{attribute 'GeneratedUsingTerminal: EL5001--0000'}
{attribute addProperty BoxType "EL5001--0000"}
{attribute addProperty Description "EL5001 1Ch. SSI Encoder"}
{attribute addProperty Physics "KK"}
{attribute addProperty Id "Channel_1AT %I*Channel_4E63E14D5WcStateAT %I*WcState_9091E0EB2InfoDataAT %I*InfoData_32EB74EA10"}
{attribute addProperty CRC "1375238614"}
{attribute addProperty Size "17"}
TYPE EL5001_51F879D6 EXTENDS EtcSlaveTerminalBase_947E5A46 :
STRUCT
	{attribute addProperty Name "Channel_1"}
	Channel_1 : Channel_4E63E14D;
	{attribute addProperty Name "WcState"}
	WcState : WcState_9091E0EB;
	{attribute addProperty Name "InfoData"}
	InfoData : InfoData_32EB74EA;
END_STRUCT
END_TYPE

(* stored: Version 1.2.0.0, ProductVersion 3.1.4024.9
   DUT EL5001_51F879D6: Id {239722e6-ec59-4625-87d0-b5d353251268} *)
